{attribute 'Tc2GvlVarNames'}
{attribute 'strict'}
//Stato Richiesta LGV
TYPE e_Stato_Richiesta_LGV_1 :
(
	NESSUNA_REQ_LGV	 	:= 0,	(* NESSUNA RICHIESTA/CHIAMATA LGV *)
	REQ_LGV			 	:= 1 	(* CHIAMATA LGV *)
);
END_TYPE

(* stored: Version 1.1.0.1, ProductVersion 3.1.4022.10
   EnumerationTextList e_Stato_Richiesta_LGV_1: Id {0cb26ea8-089b-446b-bb52-49e74504cdd0} *)
